FUNCTION_BLOCK Reset4
VAR_INPUT
END_VAR
VAR_OUTPUT
END_VAR
VAR
END_VAR

END_FUNCTION_BLOCK

(* stored: Version 1.1.0.1, ProductVersion 3.1.4024.11
   POU Reset4: Id {4d8349bd-ecc4-4b33-813c-cce1cce86081}, SpecialFunc None *)
